Staubli VAL3: teach.pgx

public program teach(num x_nConvNum (dimensions=1), tool x_tTool (dimensions=1), frame x_fFrame (dimensions=1), point& x_pLoc[] (dimensions=1), num& x_nError[] (dimensions=1))
begin
  // This program returns the coordinates of a point, in the specified
  //  frame, with respect to the instantaneous location of the conveyor.
  //  It is usually used when the detection device doesn’t provide all
  //  necessary information about the position of the object on the
  //  conveyor like for instance a sensor. A specific procedure must
  //  be performed to teach a location that way.
  //
  // Input Param
  //  x_nConvNum      : Conveyor number
  //  x_tTool         : Tool Center Point with which the location
  //                     must be taught.
  //  x_fFrame	      : The reference frame of the location to teach.
  //
  // Output param
  //  x_pLoc          : The location to teach
  //  x_nError        : Error code
  //                0 = No error
  //               -1 = No object detected, not possible to teach
  //                     anything.
  //
  //----------------------------------------------------------------
  //
  switch x_nConvNum
    case 0
      call cnv0:teach(x_tTool,x_fFrame,x_pLoc,x_nError)
    break
    case 1
      call cnv1:teach(x_tTool,x_fFrame,x_pLoc,x_nError)
    break
  endSwitch
end
